# EPICS autosave request: RigakuApp/Db/Linkam_T96_settings.req
$(P)$(T):rampLimit
$(P)$(T):rampRate
$(P)$(T):heating
$(P)$(T):lnpMode
$(P)$(T):lnpSpeed
$(P)$(T):vacuum
$(P)$(T):vacuumLimit
$(P)$(T):temperature_RBV.SCAN
$(P)$(T):heaterPower_RBV.SCAN
$(P)$(T):lnpSpeed_RBV.SCAN
$(P)$(T):pressure_RBV.SCAN
